Yaskawa INFORM job: pipe_vertical_cylinder_program.JBI

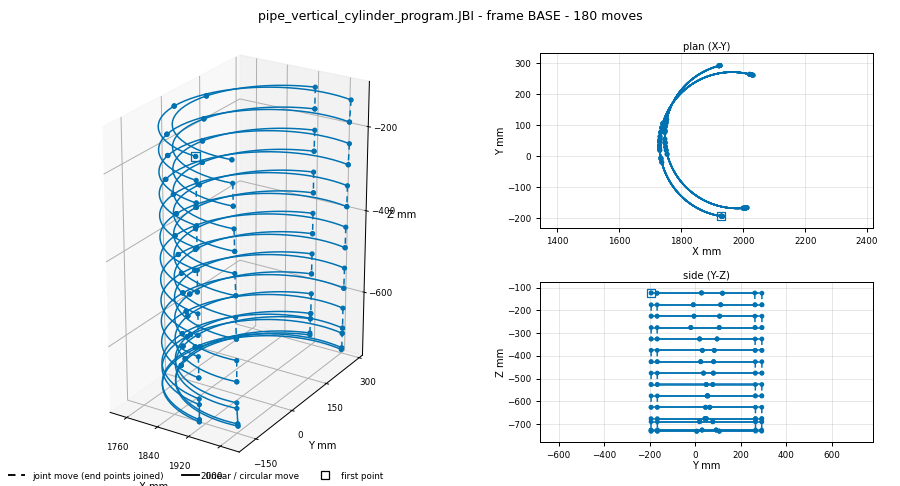
[picture p0: tool path of pipe_vertical_cylinder_program.JBI in frame BASE, 180 of 245 moves have a stored position in this frame; points joined in program order, loops and branches not executed]
/JOB
//NAME pipe_vertical_cylinder_program
//POS
///NPOS 240,0,240,0,0,0
///TOOL 0
///POSTYPE BASE
///RECTAN
///RCONF 0,0,0,0,0,0,0,0,0,0,0,0,0,0,0,0,0,0,0,0,0,0,0,0
C00000=1928.726850,-193.503248,-123.703100,-98.664603,-90.000000,5.000000
C00001=1928.726850,-193.503248,-123.703100,-98.664603,-90.000000,5.000000
C00002=1803.766355,-132.701255,-123.703100,-133.227700,-90.000000,5.000000
C00003=1730.292234,27.409491,-123.703100,-175.000000,-89.999999,5.000000
C00004=1730.292234,27.409491,-123.703100,-175.000000,-89.999999,5.000000
C00005=1730.292234,27.409491,-123.703100,-175.000000,-89.999999,5.000000
C00006=1781.666702,184.275491,-123.703100,141.204128,-90.000000,5.000000
C00007=2032.939441,261.224135,-123.703100,72.848772,-90.000000,5.000000
C00008=2029.638631,262.216252,-175.719000,73.693077,-90.000000,5.000000
C00009=2029.638631,262.216252,-175.719000,73.693077,-90.000000,5.000000
C00010=1769.062238,167.040924,-175.719000,146.436287,-90.000000,5.000000
C00011=1734.685456,-8.536686,-175.719000,-168.592181,-89.999999,5.000000
C00012=1734.685456,-8.536686,-175.719000,-168.592181,-89.999999,5.000000
C00013=1734.685456,-8.536686,-175.719000,-168.592181,-89.999999,5.000000
C00014=1817.100045,-144.317116,-175.719000,-128.894865,-90.000000,5.000000
C00015=1929.622284,-193.637929,-175.719000,-98.442790,-90.000000,5.000000
C00016=1929.392588,-193.603719,-225.637000,-98.499677,-90.000000,5.000000
C00017=1929.392588,-193.603719,-225.637000,-98.499677,-90.000000,5.000000
C00018=1818.955137,-145.798235,-225.637000,-128.313371,-90.000000,5.000000
C00019=1734.124931,-5.666309,-225.637000,-169.308593,-90.000000,5.000000
C00020=1734.124931,-5.666309,-225.637000,-169.308593,-90.000000,5.000000
C00021=1734.124931,-5.666309,-225.637000,-169.308593,-90.000000,5.000000
C00022=1767.706003,164.973175,-225.637000,147.042036,-90.000000,5.000000
C00023=2030.665258,261.913359,-225.637000,73.430878,-90.000000,5.000000
C00024=2028.642457,262.505288,-275.664500,73.947163,-89.999999,5.000000
C00025=2028.642457,262.505288,-275.664500,73.947163,-89.999999,5.000000
C00026=1774.024229,174.224845,-275.664500,144.297428,-90.000000,5.000000
C00027=1737.151101,-19.412290,-275.664500,-165.860235,-89.999999,5.000000
C00028=1737.151101,-19.412290,-275.664500,-165.860235,-89.999999,5.000000
C00029=1737.151101,-19.412290,-275.664500,-165.860235,-89.999999,5.000000
C00030=1813.642432,-141.472628,-275.664500,-129.991638,-89.999999,5.000000
C00031=1929.861431,-193.673300,-275.664500,-98.383572,-90.000000,5.000000
C00032=1930.229081,-193.727183,-325.652000,-98.292551,-90.000000,5.000000
C00033=1930.229081,-193.727183,-325.652000,-98.292551,-90.000000,5.000000
C00034=1817.110702,-144.325714,-325.652000,-128.891511,-89.999999,5.000000
C00035=1730.802620,19.160247,-325.652000,-175.000000,-89.999999,5.000000
C00036=1730.802620,19.160247,-325.652000,-175.000000,-89.999999,5.000000
C00037=1730.802620,19.160247,-325.652000,-175.000000,-89.999999,5.000000
C00038=1796.433054,200.951153,-325.652000,135.745887,-89.999999,5.000000
C00039=2027.683085,262.779127,-325.652000,74.191557,-89.999999,5.000000
C00040=2027.035362,262.961511,-375.720500,74.356393,-90.000000,5.000000
C00041=2027.035362,262.961511,-375.720500,74.356393,-90.000000,5.000000
C00042=1805.405013,209.679833,-375.720500,132.679262,-90.000000,5.000000
C00043=1730.156224,31.179849,-375.720500,-175.000000,-90.000000,5.000000
C00044=1730.156224,31.179849,-375.720500,-175.000000,-90.000000,5.000000
C00045=1730.156224,31.179849,-375.720500,-175.000000,-90.000000,5.000000
C00046=1809.670901,-138.064690,-375.720500,-131.273602,-90.000000,5.000000
C00047=1930.707197,-193.796365,-375.720500,-98.174212,-90.000000,5.000000
C00048=1930.156968,-193.716661,-425.642000,-98.310402,-90.000000,5.000000
C00049=1930.156968,-193.716661,-425.642000,-98.310402,-90.000000,5.000000
C00050=1810.851421,-139.093862,-425.642000,-130.889959,-90.000000,5.000000
C00051=1730.476143,23.857273,-425.642000,-175.000000,-89.999999,5.000000
C00052=1730.476143,23.857273,-425.642000,-175.000000,-89.999999,5.000000
C00053=1730.476143,23.857273,-425.642000,-175.000000,-89.999999,5.000000
C00054=1797.622153,202.162794,-425.642000,135.330030,-90.000000,5.000000
C00055=2025.366615,263.422150,-425.642000,74.780457,-89.999999,5.000000
C00056=2024.582475,263.634022,-475.674000,74.979427,-89.999999,5.000000
C00057=2024.582475,263.634022,-475.674000,74.979427,-89.999999,5.000000
C00058=1812.932633,216.327800,-475.674000,130.218963,-90.000000,5.000000
C00059=1730.069000,36.289969,-475.674000,-175.000000,-90.000000,5.000000
C00060=1730.069000,36.289969,-475.674000,-175.000000,-90.000000,5.000000
C00061=1730.069000,36.289969,-475.674000,-175.000000,-90.000000,5.000000
C00062=1799.181735,-128.272634,-475.674000,-134.789187,-90.000000,5.000000
C00063=1931.272436,-193.876854,-475.674000,-98.034354,-89.999999,5.000000
C00064=1931.050597,-193.845432,-525.719500,-98.089239,-90.000000,5.000000
C00065=1931.050597,-193.845432,-525.719500,-98.089239,-90.000000,5.000000
C00066=1800.469988,-129.541592,-525.719500,-134.346233,-90.000000,5.000000
C00067=1730.286568,47.914358,-525.719500,175.000000,-90.000000,5.000000
C00068=1730.286568,47.914358,-525.719500,175.000000,-90.000000,5.000000
C00069=1730.286568,47.914358,-525.719500,175.000000,-90.000000,5.000000
C00070=1804.165719,208.528758,-525.719500,133.093586,-90.000000,5.000000
C00071=2024.191048,263.738692,-525.719500,75.078680,-90.000000,5.000000
C00072=2023.212614,263.997157,-575.675000,75.326578,-89.999999,5.000000
C00073=2023.212614,263.997157,-575.675000,75.326578,-89.999999,5.000000
C00074=1825.684629,226.373546,-575.675000,126.241588,-90.000000,5.000000
C00075=1730.514547,52.227781,-575.675000,175.000000,-90.000000,5.000000
C00076=1730.514547,52.227781,-575.675000,175.000000,-90.000000,5.000000
C00077=1730.514547,52.227781,-575.675000,175.000000,-90.000000,5.000000
C00078=1793.291675,-122.210572,-575.675000,-136.859769,-90.000000,5.000000
C00079=1931.380796,-193.892123,-575.675000,-98.007548,-90.000000,5.000000
C00080=1932.261457,-194.014304,-625.648500,-97.789756,-89.999999,5.000000
C00081=1932.261457,-194.014304,-625.648500,-97.789756,-89.999999,5.000000
C00082=1795.572876,-124.610612,-625.648500,-136.048653,-90.000000,5.000000
C00083=1731.497878,63.580628,-625.648500,173.653822,-89.999999,5.000000
C00084=1731.497878,63.580628,-625.648500,173.653822,-89.999999,5.000000
C00085=1731.497878,63.580628,-625.648500,173.653822,-89.999999,5.000000
C00086=1822.597329,224.071230,-625.648500,127.184997,-90.000000,5.000000
C00087=2021.992990,264.313007,-625.648500,75.635193,-90.000000,5.000000
C00088=2021.971979,264.318387,-675.632500,75.640505,-89.999999,5.000000
C00089=2021.971979,264.318387,-675.632500,75.640505,-89.999999,5.000000
C00090=1833.386785,231.784430,-675.632500,123.935679,-90.000000,5.000000
C00091=1730.308675,48.409374,-675.632500,175.000000,-90.000000,5.000000
C00092=1730.308675,48.409374,-675.632500,175.000000,-90.000000,5.000000
C00093=1730.308675,48.409374,-675.632500,175.000000,-90.000000,5.000000
C00094=1788.874879,-117.362865,-675.632500,-138.466283,-90.000000,5.000000
C00095=1932.865499,-194.096136,-675.632500,-97.640439,-90.000000,5.000000
C00096=1932.928825,-194.104622,-725.587000,-97.624788,-90.000000,5.000000
C00097=1932.928825,-194.104622,-725.587000,-97.624788,-90.000000,5.000000
C00098=1789.994967,-118.618268,-725.587000,-138.054151,-90.000000,5.000000
C00099=1736.398051,91.788230,-725.587000,166.636237,-90.000000,5.000000
C00100=1736.398051,91.788230,-725.587000,166.636237,-90.000000,5.000000
C00101=1736.398051,91.788230,-725.587000,166.636237,-90.000000,5.000000
C00102=1842.925540,237.872887,-725.587000,121.163392,-90.000000,5.000000
C00103=2020.910815,264.587404,-725.587000,75.908671,-90.000000,5.000000
C00104=2021.296550,264.490227,-689.054960,75.811229,-89.999999,5.000000
C00105=2021.296550,264.490227,-689.054960,75.811229,-89.999999,5.000000
C00106=1833.152273,231.626426,-689.054960,124.004947,-90.000000,5.000000
C00107=1733.388096,77.016263,-689.054960,170.329761,-90.000000,5.000000
C00108=1733.388096,77.016263,-689.054960,170.329761,-90.000000,5.000000
C00109=1733.388096,77.016263,-689.054960,170.329761,-90.000000,5.000000
C00110=1783.733697,-111.357205,-689.054960,-140.402944,-90.000000,5.000000
C00111=1933.071448,-194.123670,-689.054960,-97.589541,-90.000000,5.000000
C00112=1932.727346,-194.077561,-730.492960,-97.674585,-90.000000,5.000000
C00113=1932.727346,-194.077561,-730.492960,-97.674585,-90.000000,5.000000
C00114=1784.333849,-112.079782,-730.492960,-140.172852,-90.000000,5.000000
C00115=1740.075522,105.423466,-730.492960,163.176287,-90.000000,5.000000
C00116=1740.075522,105.423466,-730.492960,163.176287,-90.000000,5.000000
C00117=1740.075522,105.423466,-730.492960,163.176287,-90.000000,5.000000
C00118=1847.805689,240.744060,-730.492960,119.776372,-89.999999,5.000000
C00119=2019.734901,264.879349,-730.492960,175.000000,-60.000000,-103.794533
C00120=1998.959667,-167.668544,-124.798050,-85.507848,-90.000000,5.000000
C00121=1998.959667,-167.668544,-124.798050,-85.507848,-90.000000,5.000000
C00122=1767.990520,-31.899354,-124.798050,-155.388214,-90.000000,5.000000
C00123=1753.066612,119.541293,-124.798050,166.644439,-90.000000,5.000000
C00124=1753.066612,119.541293,-124.798050,166.644439,-90.000000,5.000000
C00125=1753.066612,119.541293,-124.798050,166.644439,-90.000000,5.000000
C00126=1817.164152,232.797683,-124.798050,134.340113,-89.999999,5.000000
C00127=1925.257474,292.760021,-124.798050,103.696561,-90.000000,5.000000
C00128=1924.932131,292.680485,-175.656000,103.778603,-90.000000,5.000000
C00129=1924.932131,292.680485,-175.656000,103.778603,-90.000000,5.000000
C00130=1817.319673,232.949521,-175.656000,134.286871,-90.000000,5.000000
C00131=1751.297881,111.457631,-175.656000,168.671559,-90.000000,5.000000
C00132=1751.297881,111.457631,-175.656000,168.671559,-90.000000,5.000000
C00133=1751.297881,111.457631,-175.656000,168.671559,-90.000000,5.000000
C00134=1779.620919,-54.071017,-175.656000,-149.252249,-90.000000,5.000000
C00135=2000.839312,-167.513244,-175.656000,-85.045841,-89.999999,5.000000
C00136=2001.925642,-167.416526,-225.676500,-84.778682,-90.000000,5.000000
C00137=2001.925642,-167.416526,-225.676500,-84.778682,-90.000000,5.000000
C00138=1776.474314,-48.615748,-225.676500,-150.794977,-90.000000,5.000000
C00139=1750.392034,106.678507,-225.676500,169.863115,-90.000000,5.000000
C00140=1750.392034,106.678507,-225.676500,169.863115,-90.000000,5.000000
C00141=1750.392034,106.678507,-225.676500,169.863115,-90.000000,5.000000
C00142=1816.210959,231.860859,-225.676500,134.667500,-90.000000,5.000000
C00143=1925.502504,292.819598,-225.676500,103.634790,-90.000000,5.000000
C00144=1924.682080,292.619020,-275.719500,103.841679,-90.000000,5.000000
C00145=1924.682080,292.619020,-275.719500,103.841679,-90.000000,5.000000
C00146=1810.632436,226.155325,-275.719500,136.622257,-90.000000,5.000000
C00147=1750.118437,105.117754,-275.719500,170.251266,-90.000000,5.000000
C00148=1750.118437,105.117754,-275.719500,170.251266,-90.000000,5.000000
C00149=1750.118437,105.117754,-275.719500,170.251266,-90.000000,5.000000
C00150=1783.735100,-60.730735,-275.719500,-147.334607,-89.999999,5.000000
C00151=2003.640188,-167.253479,-275.719500,-84.356792,-90.000000,5.000000
C00152=2005.043198,-167.110573,-325.670500,-84.011333,-90.000000,5.000000
C00153=2005.043198,-167.110573,-325.670500,-84.011333,-90.000000,5.000000
C00154=1792.364461,-73.272320,-325.670500,-143.604793,-90.000000,5.000000
C00155=1748.699093,95.714976,-325.670500,172.580818,-89.999999,5.000000
C00156=1748.699093,95.714976,-325.670500,172.580818,-89.999999,5.000000
C00157=1748.699093,95.714976,-325.670500,172.580818,-89.999999,5.000000
C00158=1810.475634,225.989220,-325.670500,136.678212,-90.000000,5.000000
C00159=1924.283815,292.520519,-325.670500,103.942177,-90.000000,5.000000
C00160=1924.540718,292.584142,-375.743500,103.877345,-90.000000,5.000000
C00161=1924.540718,292.584142,-375.743500,103.877345,-90.000000,5.000000
C00162=1801.064263,215.383277,-375.743500,140.152159,-90.000000,5.000000
C00163=1747.439635,83.578278,-375.743500,175.000000,-90.000000,5.000000
C00164=1747.439635,83.578278,-375.743500,175.000000,-90.000000,5.000000
C00165=1747.439635,83.578278,-375.743500,175.000000,-90.000000,5.000000
C00166=1801.123272,-84.429686,-375.743500,-140.129604,-90.000000,5.000000
C00167=2005.299172,-167.083577,-375.743500,-83.948282,-90.000000,5.000000
C00168=2007.681799,-166.818624,-425.656500,-83.361035,-90.000000,5.000000
C00169=2007.681799,-166.818624,-425.656500,-83.361035,-90.000000,5.000000
C00170=1802.417989,-85.966312,-425.656500,-139.637393,-89.999999,5.000000
C00171=1747.231813,80.658557,-425.656500,175.000000,-90.000000,5.000000
C00172=1747.231813,80.658557,-425.656500,175.000000,-90.000000,5.000000
C00173=1747.231813,80.658557,-425.656500,175.000000,-90.000000,5.000000
C00174=1804.741959,219.683094,-425.656500,138.766126,-89.999999,5.000000
C00175=1924.217009,292.503923,-425.656500,103.959039,-89.999999,5.000000
C00176=1924.014985,292.453611,-475.660500,104.010039,-89.999999,5.000000
C00177=1924.014985,292.453611,-475.660500,104.010039,-89.999999,5.000000
C00178=1804.589067,219.508481,-475.660500,138.822978,-90.000000,5.000000
C00179=1747.163751,79.570475,-475.660500,175.000000,-90.000000,5.000000
C00180=1747.163751,79.570475,-475.660500,175.000000,-90.000000,5.000000
C00181=1747.163751,79.570475,-475.660500,175.000000,-90.000000,5.000000
C00182=1803.164428,-86.840176,-475.660500,-139.355869,-90.000000,5.000000
C00183=2007.110595,-166.884397,-475.660500,-83.501882,-90.000000,5.000000
C00184=2008.839212,-166.680986,-525.651000,-83.075518,-90.000000,5.000000
C00185=2008.839212,-166.680986,-525.651000,-83.075518,-90.000000,5.000000
C00186=1812.215183,-96.789707,-525.651000,-136.060651,-90.000000,5.000000
C00187=1747.024314,77.023291,-525.651000,175.000000,-90.000000,5.000000
C00188=1747.024314,77.023291,-525.651000,175.000000,-90.000000,5.000000
C00189=1747.024314,77.023291,-525.651000,175.000000,-90.000000,5.000000
C00190=1804.577289,219.495015,-525.651000,138.827360,-90.000000,5.000000
C00191=1923.549770,292.337027,-525.651000,104.127521,-90.000000,5.000000
C00192=1922.961564,292.188168,-575.624500,104.276150,-89.999999,5.000000
C00193=1922.961564,292.188168,-575.624500,104.276150,-89.999999,5.000000
C00194=1798.996731,212.870635,-575.624500,140.949245,-90.000000,5.000000
C00195=1746.966709,55.236508,-575.624500,-175.000000,-90.000000,5.000000
C00196=1746.966709,55.236508,-575.624500,-175.000000,-90.000000,5.000000
C00197=1746.966709,55.236508,-575.624500,-175.000000,-90.000000,5.000000
C00198=1829.345775,-112.866304,-575.624500,-130.303436,-90.000000,5.000000
C00199=2009.573435,-166.590638,-575.624500,-82.894307,-90.000000,5.000000
C00200=2009.608838,-166.586222,-625.632500,-82.885567,-90.000000,5.000000
C00201=2009.608838,-166.586222,-625.632500,-82.885567,-90.000000,5.000000
C00202=1821.838073,-106.216594,-625.632500,-132.760363,-90.000000,5.000000
C00203=1747.621232,45.237784,-625.632500,-175.000000,-90.000000,5.000000
C00204=1747.621232,45.237784,-625.632500,-175.000000,-90.000000,5.000000
C00205=1747.621232,45.237784,-625.632500,-175.000000,-90.000000,5.000000
C00206=1794.015447,206.508872,-625.632500,142.928597,-90.000000,5.000000
C00207=1923.063279,292.214025,-625.632500,104.250442,-90.000000,5.000000
C00208=1922.513675,292.073729,-675.682500,104.389390,-89.999999,5.000000
C00209=1922.513675,292.073729,-675.682500,104.389390,-89.999999,5.000000
C00210=1788.388676,198.734621,-675.682500,145.279599,-90.000000,5.000000
C00211=1747.900420,42.250925,-675.682500,-174.292516,-90.000000,5.000000
C00212=1747.900420,42.250925,-675.682500,-174.292516,-90.000000,5.000000
C00213=1747.900420,42.250925,-675.682500,-174.292516,-90.000000,5.000000
C00214=1839.134852,-120.727240,-675.682500,-127.227678,-90.000000,5.000000
C00215=2009.668320,-166.578790,-675.682500,-82.870883,-90.000000,5.000000
C00216=2011.743051,-166.309869,-725.700000,-82.358406,-90.000000,5.000000
C00217=2011.743051,-166.309869,-725.700000,-82.358406,-90.000000,5.000000
C00218=1833.832967,-116.577144,-725.700000,-128.877046,-89.999999,5.000000
C00219=1749.432997,30.126859,-725.700000,-171.298639,-90.000000,5.000000
C00220=1749.432997,30.126859,-725.700000,-171.298639,-90.000000,5.000000
C00221=1749.432997,30.126859,-725.700000,-171.298639,-90.000000,5.000000
C00222=1787.619822,197.618204,-725.700000,145.611655,-90.000000,5.000000
C00223=1921.110199,291.709014,-725.700000,104.744603,-89.999999,5.000000
C00224=1921.946227,291.927387,-689.010460,104.532939,-90.000000,5.000000
C00225=1921.946227,291.927387,-689.010460,104.532939,-90.000000,5.000000
C00226=1786.725932,196.302565,-689.010460,146.001283,-89.999999,5.000000
C00227=1751.390250,19.107946,-689.010460,-168.556942,-90.000000,5.000000
C00228=1751.390250,19.107946,-689.010460,-168.556942,-90.000000,5.000000
C00229=1751.390250,19.107946,-689.010460,-168.556942,-90.000000,5.000000
C00230=1839.368673,-120.904666,-689.010460,-127.155779,-90.000000,5.000000
C00231=2009.928458,-166.546106,-689.010460,-82.806659,-89.999999,5.000000
C00232=2012.523618,-166.203804,-730.753960,-82.165441,-89.999999,5.000000
C00233=2012.523618,-166.203804,-730.753960,-82.165441,-89.999999,5.000000
C00234=1852.025431,-129.851901,-730.753960,-123.358242,-90.000000,5.000000
C00235=1754.324738,6.434227,-730.753960,-165.369853,-90.000000,5.000000
C00236=1754.324738,6.434227,-730.753960,-165.369853,-90.000000,5.000000
C00237=1754.324738,6.434227,-730.753960,-165.369853,-90.000000,5.000000
C00238=1784.258203,192.567208,-730.753960,147.097956,-90.000000,5.000000
C00239=1921.499557,291.811126,-730.753960,175.000000,-60.000000,-75.353999
///POSTYPE PULSE
///PULSE
EX00000=147456.0
EX00001=354304.0
///POSTYPE PULSE
///PULSE
EC00000=147456.0
EC00001=147456.0
EC00002=147456.0
EC00003=147456.0
EC00004=147456.0
EC00005=147456.0
EC00006=147456.0
EC00007=147456.0
EC00008=147456.0
EC00009=147456.0
EC00010=147456.0
EC00011=147456.0
EC00012=147456.0
EC00013=147456.0
EC00014=147456.0
EC00015=147456.0
EC00016=147456.0
EC00017=147456.0
EC00018=147456.0
EC00019=147456.0
EC00020=147456.0
EC00021=147456.0
EC00022=147456.0
EC00023=147456.0
EC00024=147456.0
EC00025=147456.0
EC00026=147456.0
EC00027=147456.0
EC00028=147456.0
EC00029=147456.0
EC00030=147456.0
EC00031=147456.0
EC00032=147456.0
EC00033=147456.0
EC00034=147456.0
EC00035=147456.0
EC00036=147456.0
EC00037=147456.0
EC00038=147456.0
EC00039=147456.0
EC00040=147456.0
EC00041=147456.0
EC00042=147456.0
EC00043=147456.0
EC00044=147456.0
EC00045=147456.0
EC00046=147456.0
EC00047=147456.0
EC00048=147456.0
EC00049=147456.0
EC00050=147456.0
EC00051=147456.0
EC00052=147456.0
EC00053=147456.0
EC00054=147456.0
EC00055=147456.0
EC00056=147456.0
EC00057=147456.0
EC00058=147456.0
EC00059=147456.0
EC00060=147456.0
EC00061=147456.0
EC00062=147456.0
EC00063=147456.0
EC00064=147456.0
EC00065=147456.0
EC00066=147456.0
EC00067=147456.0
EC00068=147456.0
EC00069=147456.0
EC00070=147456.0
EC00071=147456.0
EC00072=147456.0
EC00073=147456.0
EC00074=147456.0
EC00075=147456.0
EC00076=147456.0
EC00077=147456.0
EC00078=147456.0
EC00079=147456.0
EC00080=147456.0
EC00081=147456.0
EC00082=147456.0
EC00083=147456.0
EC00084=147456.0
EC00085=147456.0
EC00086=147456.0
EC00087=147456.0
EC00088=147456.0
EC00089=147456.0
EC00090=147456.0
EC00091=147456.0
EC00092=147456.0
EC00093=147456.0
EC00094=147456.0
EC00095=147456.0
EC00096=147456.0
EC00097=147456.0
EC00098=147456.0
EC00099=147456.0
EC00100=147456.0
EC00101=147456.0
EC00102=147456.0
EC00103=147456.0
EC00104=147456.0
EC00105=147456.0
EC00106=147456.0
EC00107=147456.0
EC00108=147456.0
EC00109=147456.0
EC00110=147456.0
EC00111=147456.0
EC00112=147456.0
EC00113=147456.0
EC00114=147456.0
EC00115=147456.0
EC00116=147456.0
EC00117=147456.0
EC00118=147456.0
EC00119=147456.0
EC00120=354304.0
EC00121=354304.0
EC00122=354304.0
EC00123=354304.0
EC00124=354304.0
EC00125=354304.0
EC00126=354304.0
EC00127=354304.0
EC00128=354304.0
EC00129=354304.0
EC00130=354304.0
EC00131=354304.0
EC00132=354304.0
EC00133=354304.0
EC00134=354304.0
EC00135=354304.0
EC00136=354304.0
EC00137=354304.0
EC00138=354304.0
EC00139=354304.0
EC00140=354304.0
EC00141=354304.0
EC00142=354304.0
EC00143=354304.0
EC00144=354304.0
EC00145=354304.0
EC00146=354304.0
EC00147=354304.0
EC00148=354304.0
EC00149=354304.0
EC00150=354304.0
EC00151=354304.0
EC00152=354304.0
EC00153=354304.0
EC00154=354304.0
EC00155=354304.0
EC00156=354304.0
EC00157=354304.0
EC00158=354304.0
EC00159=354304.0
EC00160=354304.0
EC00161=354304.0
EC00162=354304.0
EC00163=354304.0
EC00164=354304.0
EC00165=354304.0
EC00166=354304.0
EC00167=354304.0
EC00168=354304.0
EC00169=354304.0
EC00170=354304.0
EC00171=354304.0
EC00172=354304.0
EC00173=354304.0
EC00174=354304.0
EC00175=354304.0
EC00176=354304.0
EC00177=354304.0
EC00178=354304.0
EC00179=354304.0
EC00180=354304.0
EC00181=354304.0
EC00182=354304.0
EC00183=354304.0
EC00184=354304.0
EC00185=354304.0
EC00186=354304.0
EC00187=354304.0
EC00188=354304.0
EC00189=354304.0
EC00190=354304.0
EC00191=354304.0
EC00192=354304.0
EC00193=354304.0
EC00194=354304.0
EC00195=354304.0
EC00196=354304.0
EC00197=354304.0
EC00198=354304.0
EC00199=354304.0
EC00200=354304.0
EC00201=354304.0
EC00202=354304.0
EC00203=354304.0
EC00204=354304.0
EC00205=354304.0
EC00206=354304.0
EC00207=354304.0
EC00208=354304.0
EC00209=354304.0
EC00210=354304.0
EC00211=354304.0
EC00212=354304.0
EC00213=354304.0
EC00214=354304.0
EC00215=354304.0
EC00216=354304.0
EC00217=354304.0
EC00218=354304.0
EC00219=354304.0
EC00220=354304.0
EC00221=354304.0
EC00222=354304.0
EC00223=354304.0
EC00224=354304.0
EC00225=354304.0
EC00226=354304.0
EC00227=354304.0
EC00228=354304.0
EC00229=354304.0
EC00230=354304.0
EC00231=354304.0
EC00232=354304.0
EC00233=354304.0
EC00234=354304.0
EC00235=354304.0
EC00236=354304.0
EC00237=354304.0
EC00238=354304.0
EC00239=354304.0
//INST
///DATE 2023/08/15 13:38
///ATTR SC,RW,RJ
////FRAME BASE
///GROUP1 RB1,ST1
NOP
MOVJ P009 EX000 VJ=15.00
MOVJ C00000 EC00000 VJ=15.0
CALL JOB:SPYON
MOVC C00001 EC00001 V=150.0
MOVC C00002 EC00002 V=150.0
MOVC C00003 EC00003 V=150.0
MOVJ C00004 EC00004 VJ=15.0
MOVC C00005 EC00005 V=150.0
MOVC C00006 EC00006 V=150.0
MOVC C00007 EC00007 V=150.0
MOVJ C00008 EC00008 VJ=15.0
MOVC C00009 EC00009 V=150.0
MOVC C00010 EC00010 V=150.0
MOVC C00011 EC00011 V=150.0
MOVJ C00012 EC00012 VJ=15.0
MOVC C00013 EC00013 V=150.0
MOVC C00014 EC00014 V=150.0
MOVC C00015 EC00015 V=150.0
MOVJ C00016 EC00016 VJ=15.0
MOVC C00017 EC00017 V=150.0
MOVC C00018 EC00018 V=150.0
MOVC C00019 EC00019 V=150.0
MOVJ C00020 EC00020 VJ=15.0
MOVC C00021 EC00021 V=150.0
MOVC C00022 EC00022 V=150.0
MOVC C00023 EC00023 V=150.0
MOVJ C00024 EC00024 VJ=15.0
MOVC C00025 EC00025 V=150.0
MOVC C00026 EC00026 V=150.0
MOVC C00027 EC00027 V=150.0
MOVJ C00028 EC00028 VJ=15.0
MOVC C00029 EC00029 V=150.0
MOVC C00030 EC00030 V=150.0
MOVC C00031 EC00031 V=150.0
MOVJ C00032 EC00032 VJ=15.0
MOVC C00033 EC00033 V=150.0
MOVC C00034 EC00034 V=150.0
MOVC C00035 EC00035 V=150.0
MOVJ C00036 EC00036 VJ=15.0
MOVC C00037 EC00037 V=150.0
MOVC C00038 EC00038 V=150.0
MOVC C00039 EC00039 V=150.0
MOVJ C00040 EC00040 VJ=15.0
MOVC C00041 EC00041 V=150.0
MOVC C00042 EC00042 V=150.0
MOVC C00043 EC00043 V=150.0
MOVJ C00044 EC00044 VJ=15.0
MOVC C00045 EC00045 V=150.0
MOVC C00046 EC00046 V=150.0
MOVC C00047 EC00047 V=150.0
MOVJ C00048 EC00048 VJ=15.0
MOVC C00049 EC00049 V=150.0
MOVC C00050 EC00050 V=150.0
MOVC C00051 EC00051 V=150.0
MOVJ C00052 EC00052 VJ=15.0
MOVC C00053 EC00053 V=150.0
MOVC C00054 EC00054 V=150.0
MOVC C00055 EC00055 V=150.0
MOVJ C00056 EC00056 VJ=15.0
MOVC C00057 EC00057 V=150.0
MOVC C00058 EC00058 V=150.0
MOVC C00059 EC00059 V=150.0
MOVJ C00060 EC00060 VJ=15.0
MOVC C00061 EC00061 V=150.0
MOVC C00062 EC00062 V=150.0
MOVC C00063 EC00063 V=150.0
MOVJ C00064 EC00064 VJ=15.0
MOVC C00065 EC00065 V=150.0
MOVC C00066 EC00066 V=150.0
MOVC C00067 EC00067 V=150.0
MOVJ C00068 EC00068 VJ=15.0
MOVC C00069 EC00069 V=150.0
MOVC C00070 EC00070 V=150.0
MOVC C00071 EC00071 V=150.0
MOVJ C00072 EC00072 VJ=15.0
MOVC C00073 EC00073 V=150.0
MOVC C00074 EC00074 V=150.0
MOVC C00075 EC00075 V=150.0
MOVJ C00076 EC00076 VJ=15.0
MOVC C00077 EC00077 V=150.0
MOVC C00078 EC00078 V=150.0
MOVC C00079 EC00079 V=150.0
MOVJ C00080 EC00080 VJ=15.0
MOVC C00081 EC00081 V=150.0
MOVC C00082 EC00082 V=150.0
MOVC C00083 EC00083 V=150.0
MOVJ C00084 EC00084 VJ=15.0
MOVC C00085 EC00085 V=150.0
MOVC C00086 EC00086 V=150.0
MOVC C00087 EC00087 V=150.0
MOVJ C00088 EC00088 VJ=15.0
MOVC C00089 EC00089 V=150.0
MOVC C00090 EC00090 V=150.0
MOVC C00091 EC00091 V=150.0
MOVJ C00092 EC00092 VJ=15.0
MOVC C00093 EC00093 V=150.0
MOVC C00094 EC00094 V=150.0
MOVC C00095 EC00095 V=150.0
MOVJ C00096 EC00096 VJ=15.0
MOVC C00097 EC00097 V=150.0
MOVC C00098 EC00098 V=150.0
MOVC C00099 EC00099 V=150.0
MOVJ C00100 EC00100 VJ=15.0
MOVC C00101 EC00101 V=150.0
MOVC C00102 EC00102 V=150.0
MOVC C00103 EC00103 V=150.0
MOVJ C00104 EC00104 VJ=15.0
MOVC C00105 EC00105 V=150.0
MOVC C00106 EC00106 V=150.0
MOVC C00107 EC00107 V=150.0
MOVJ C00108 EC00108 VJ=15.0
MOVC C00109 EC00109 V=150.0
MOVC C00110 EC00110 V=150.0
MOVC C00111 EC00111 V=150.0
MOVJ C00112 EC00112 VJ=15.0
MOVC C00113 EC00113 V=150.0
MOVC C00114 EC00114 V=150.0
MOVC C00115 EC00115 V=150.0
MOVJ C00116 EC00116 VJ=15.0
MOVC C00117 EC00117 V=150.0
MOVC C00118 EC00118 V=150.0
MOVC C00119 EC00119 V=150.0
CALL JOB:SPYOF
MOVJ P009 VJ=15.00
MOVL P009 EX00000 V=150.0
MOVJ C00120 EC00120 VJ=15.0
CALL JOB:SPYON
MOVC C00121 EC00121 V=150.0
MOVC C00122 EC00122 V=150.0
MOVC C00123 EC00123 V=150.0
MOVJ C00124 EC00124 VJ=15.0
MOVC C00125 EC00125 V=150.0
MOVC C00126 EC00126 V=150.0
MOVC C00127 EC00127 V=150.0
MOVJ C00128 EC00128 VJ=15.0
MOVC C00129 EC00129 V=150.0
MOVC C00130 EC00130 V=150.0
MOVC C00131 EC00131 V=150.0
MOVJ C00132 EC00132 VJ=15.0
MOVC C00133 EC00133 V=150.0
MOVC C00134 EC00134 V=150.0
MOVC C00135 EC00135 V=150.0
MOVJ C00136 EC00136 VJ=15.0
MOVC C00137 EC00137 V=150.0
MOVC C00138 EC00138 V=150.0
MOVC C00139 EC00139 V=150.0
MOVJ C00140 EC00140 VJ=15.0
MOVC C00141 EC00141 V=150.0
MOVC C00142 EC00142 V=150.0
MOVC C00143 EC00143 V=150.0
MOVJ C00144 EC00144 VJ=15.0
MOVC C00145 EC00145 V=150.0
MOVC C00146 EC00146 V=150.0
MOVC C00147 EC00147 V=150.0
MOVJ C00148 EC00148 VJ=15.0
MOVC C00149 EC00149 V=150.0
MOVC C00150 EC00150 V=150.0
MOVC C00151 EC00151 V=150.0
MOVJ C00152 EC00152 VJ=15.0
MOVC C00153 EC00153 V=150.0
MOVC C00154 EC00154 V=150.0
MOVC C00155 EC00155 V=150.0
MOVJ C00156 EC00156 VJ=15.0
MOVC C00157 EC00157 V=150.0
MOVC C00158 EC00158 V=150.0
MOVC C00159 EC00159 V=150.0
MOVJ C00160 EC00160 VJ=15.0
MOVC C00161 EC00161 V=150.0
MOVC C00162 EC00162 V=150.0
MOVC C00163 EC00163 V=150.0
MOVJ C00164 EC00164 VJ=15.0
MOVC C00165 EC00165 V=150.0
MOVC C00166 EC00166 V=150.0
MOVC C00167 EC00167 V=150.0
MOVJ C00168 EC00168 VJ=15.0
MOVC C00169 EC00169 V=150.0
MOVC C00170 EC00170 V=150.0
MOVC C00171 EC00171 V=150.0
MOVJ C00172 EC00172 VJ=15.0
MOVC C00173 EC00173 V=150.0
MOVC C00174 EC00174 V=150.0
MOVC C00175 EC00175 V=150.0
MOVJ C00176 EC00176 VJ=15.0
MOVC C00177 EC00177 V=150.0
MOVC C00178 EC00178 V=150.0
MOVC C00179 EC00179 V=150.0
MOVJ C00180 EC00180 VJ=15.0
MOVC C00181 EC00181 V=150.0
MOVC C00182 EC00182 V=150.0
MOVC C00183 EC00183 V=150.0
MOVJ C00184 EC00184 VJ=15.0
MOVC C00185 EC00185 V=150.0
MOVC C00186 EC00186 V=150.0
MOVC C00187 EC00187 V=150.0
MOVJ C00188 EC00188 VJ=15.0
MOVC C00189 EC00189 V=150.0
MOVC C00190 EC00190 V=150.0
MOVC C00191 EC00191 V=150.0
MOVJ C00192 EC00192 VJ=15.0
MOVC C00193 EC00193 V=150.0
MOVC C00194 EC00194 V=150.0
MOVC C00195 EC00195 V=150.0
MOVJ C00196 EC00196 VJ=15.0
MOVC C00197 EC00197 V=150.0
MOVC C00198 EC00198 V=150.0
MOVC C00199 EC00199 V=150.0
MOVJ C00200 EC00200 VJ=15.0
MOVC C00201 EC00201 V=150.0
MOVC C00202 EC00202 V=150.0
MOVC C00203 EC00203 V=150.0
MOVJ C00204 EC00204 VJ=15.0
MOVC C00205 EC00205 V=150.0
MOVC C00206 EC00206 V=150.0
MOVC C00207 EC00207 V=150.0
MOVJ C00208 EC00208 VJ=15.0
MOVC C00209 EC00209 V=150.0
MOVC C00210 EC00210 V=150.0
MOVC C00211 EC00211 V=150.0
MOVJ C00212 EC00212 VJ=15.0
MOVC C00213 EC00213 V=150.0
MOVC C00214 EC00214 V=150.0
MOVC C00215 EC00215 V=150.0
MOVJ C00216 EC00216 VJ=15.0
MOVC C00217 EC00217 V=150.0
MOVC C00218 EC00218 V=150.0
MOVC C00219 EC00219 V=150.0
MOVJ C00220 EC00220 VJ=15.0
MOVC C00221 EC00221 V=150.0
MOVC C00222 EC00222 V=150.0
MOVC C00223 EC00223 V=150.0
MOVJ C00224 EC00224 VJ=15.0
MOVC C00225 EC00225 V=150.0
MOVC C00226 EC00226 V=150.0
MOVC C00227 EC00227 V=150.0
MOVJ C00228 EC00228 VJ=15.0
MOVC C00229 EC00229 V=150.0
MOVC C00230 EC00230 V=150.0
MOVC C00231 EC00231 V=150.0
MOVJ C00232 EC00232 VJ=15.0
MOVC C00233 EC00233 V=150.0
MOVC C00234 EC00234 V=150.0
MOVC C00235 EC00235 V=150.0
MOVJ C00236 EC00236 VJ=15.0
MOVC C00237 EC00237 V=150.0
MOVC C00238 EC00238 V=150.0
MOVC C00239 EC00239 V=150.0
CALL JOB:SPYOF
MOVJ P009 VJ=15.00
MOVL P009 EX00001 V=150.0
END
